// TIA Portal V18 export
TYPE "UTD_AHUsAO"
// stored: IsFailsafeCompliant false
   STRUCT
      rSAFAnalog : Array[1..3] of Real;
      rHeater : Array[1..3] of Real;
      rMixingAirDumper : Array[1..3] of Real;
      rExtractAirDumper : Array[1..3] of Real;
      rCooler : Array[1..3] of Real;
      rWHU : Array[1..3] of Real;
   END_STRUCT;
END_TYPE
